INTERFACE If_Parameters

PROPERTY Par : REFERENCE TO dt_Parameters
GET
END_GET
END_PROPERTY

END_INTERFACE

(* stored: Version 1.1.0.1, ProductVersion 3.1.4024.15
   Itf If_Parameters: Id {992d696a-cb09-44dd-8546-b18a5a1eeee3}
   Property Par: Id {bc6e99ad-5d59-496f-a8dc-a1d3efdbedb7}
   Get Get: Id {c02b2cab-888c-4985-a0bc-f4dd54aaca49} *)
